PROGRAM PRG_Filters_TEST
VAR
END_VAR

END_PROGRAM

(* stored: Version 1.1.0.1, ProductVersion 3.1.4024.13
   POU PRG_Filters_TEST: Id {592f1f20-45ca-45e5-8cc6-b4ce6d2832b4}, SpecialFunc None *)
